(* Logix 5000 project; controller cal1632 1756-L62 rev 16.20; software revision 16.05; part 13 of 57 *)
(* tags used below, declared in another part *)
   AFI : BOOL;
   FAULT : BOOL;
   p01_param_fan_zero_speed : REAL;
   p01_param_open_oven_exh_sp : REAL;
   p01_param_open_oven_recirc_sp : REAL;
   p01_recipe_active : recipe;
   p01r02 : routine;
   p01r09_open_oven : BOOL;
   p01r09_pb_global_reset : BOOL;
   p02_dint_from_hmi : hmi_dint;
   p11_ai_exh_rpm : REAL;
   p11_ai_lfl : REAL;
   p11_ai_recirc_rpm : REAL;
   p11_ao_exhaust_selected_speed : REAL;
   p11_ao_recirc_selected_speed : REAL;
   p11_di_burner_auto : BOOL;
   p11_di_door_open : BOOL;
   p11_di_exh : acs800_di_normal;
   p11_di_exh_fan_mtr_ts : BOOL;
   p11_di_exh_flow_ok : BOOL;
   p11_di_flame_on : BOOL;
   p11_di_fresh_air_clean : BOOL;
   p11_di_recirc : acs800_di_normal;
   p11_di_recirc_fan_mtr_ts : BOOL;
   p11_di_recirc_flow_ok : BOOL;
   p11_di_sp00 : BOOL;
   p11_di_tc01_bo : BOOL;
   p11_di_tc02_bo : BOOL;
   p11_di_zone_air_clean : BOOL;
   p11_do_enable_burner : BOOL;
   p11_do_exh : acs800_do_normal;
   p11_do_recirc : acs800_do_normal;
   p11_param_lfl_hl : REAL;
   p11_param_tc01_dev : REAL;
   p11r02_shutdown_temp : BOOL;
   p11r20_safeties_ok : BOOL;
   p11r20_state : DINT;
   p11r30 : routine;
   p11r30_pb_zone_on : BOOL;
   p11r30_pid_temp_sp_error : REAL;
   p11r30_request_deviation_warning : BOOL;
   p11r30_request_heat : BOOL;
   p11r30_request_heat_last : BOOL;
   p11r30_request_manual : BOOL;
   p11r30_timer_fault : TIMER[16];
   p11r30_timer_warning : TIMER[12];
   p11r31 : routine;
   p11r31_pb_start : BOOL;
   p11r31_pb_stop : BOOL;
   p11r31_request_auto_run : BOOL;
   p11r31_run_permissive : BOOL;
   p11r31_timer_fault : TIMER[5];
   p11r31_timer_warning : TIMER[5];
   p11r31_vfd_stopped : BOOL;
   p11r32 : routine;
   p11r32_pb_start : BOOL;
   p11r32_pb_stop : BOOL;
   p11r32_request_auto_run : BOOL;
   p11r32_run_permissive : BOOL;
   p11r32_timer_fault : TIMER[5];
   p11r32_timer_warning : TIMER[5];
   p11r32_vfd_stopped : BOOL;
   p12r30 : routine;
   p23_di_exhaust_speed_ok : BOOL;
   p23_di_supply_speed_ok : BOOL;
   p23r02 : routine;
(* P11_Zone_1, continued *)

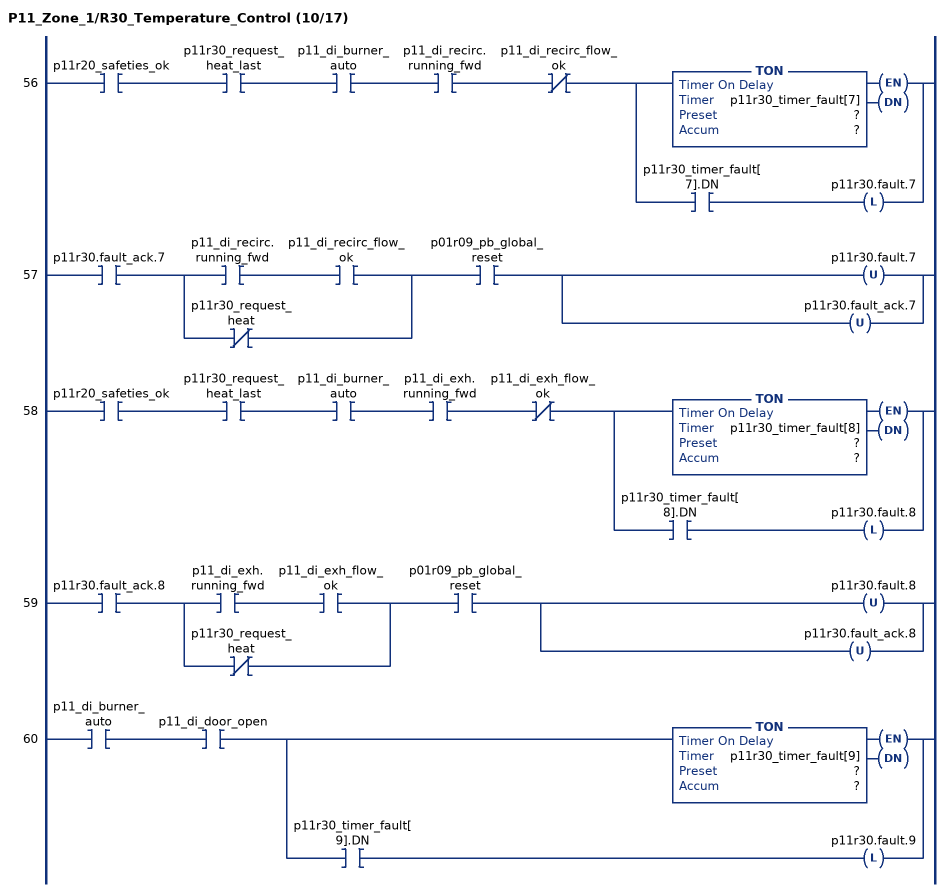
   [picture p239: P11_Zone_1/R30_Temperature_Control rungs 56-60]
   56: XIC(p11r20_safeties_ok)XIC(p11r30_request_heat_last)XIC(p11_di_burner_auto)XIC(p11_di_recirc.running_fwd)XIO(p11_di_recirc_flow_ok)[TON(p11r30_timer_fault[7],?,?) ,XIC(p11r30_timer_fault[7].DN) OTL(p11r30.fault.7) ];
   57: XIC(p11r30.fault_ack.7)[XIC(p11_di_recirc.running_fwd) XIC(p11_di_recirc_flow_ok) ,XIO(p11r30_request_heat) ]XIC(p01r09_pb_global_reset)[OTU(p11r30.fault.7) ,OTU(p11r30.fault_ack.7) ];
   58: XIC(p11r20_safeties_ok)XIC(p11r30_request_heat_last)XIC(p11_di_burner_auto)XIC(p11_di_exh.running_fwd)XIO(p11_di_exh_flow_ok)[TON(p11r30_timer_fault[8],?,?) ,XIC(p11r30_timer_fault[8].DN) OTL(p11r30.fault.8) ];
   59: XIC(p11r30.fault_ack.8)[XIC(p11_di_exh.running_fwd) XIC(p11_di_exh_flow_ok) ,XIO(p11r30_request_heat) ]XIC(p01r09_pb_global_reset)[OTU(p11r30.fault.8) ,OTU(p11r30.fault_ack.8) ];
   60: XIC(p11_di_burner_auto)XIC(p11_di_door_open)[TON(p11r30_timer_fault[9],?,?) ,XIC(p11r30_timer_fault[9].DN) OTL(p11r30.fault.9) ];
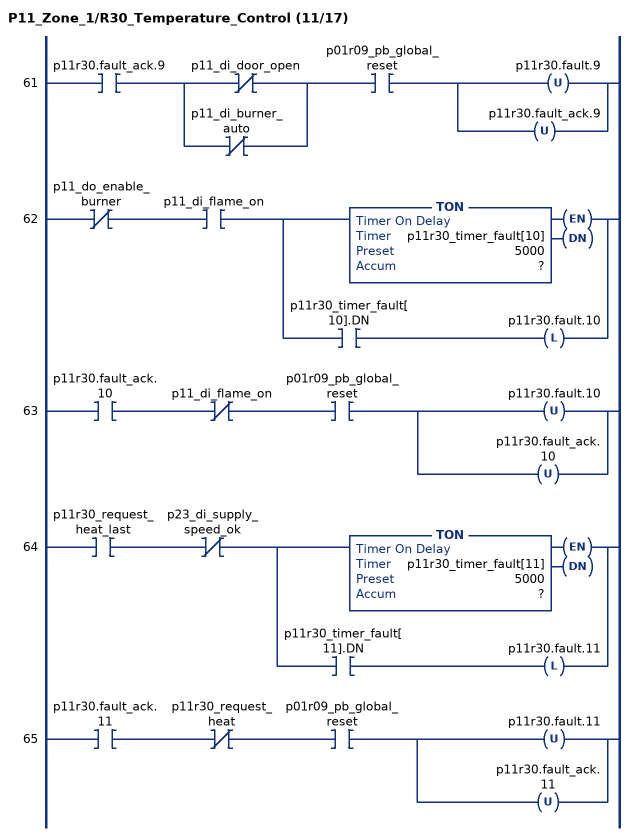
   61: XIC(p11r30.fault_ack.9)[XIO(p11_di_door_open) ,XIO(p11_di_burner_auto) ]XIC(p01r09_pb_global_reset)[OTU(p11r30.fault.9) ,OTU(p11r30.fault_ack.9) ];
   62: XIO(p11_do_enable_burner)XIC(p11_di_flame_on)[TON(p11r30_timer_fault[10],?,?) ,XIC(p11r30_timer_fault[10].DN) OTL(p11r30.fault.10) ];
   63: XIC(p11r30.fault_ack.10)XIO(p11_di_flame_on)XIC(p01r09_pb_global_reset)[OTU(p11r30.fault.10) ,OTU(p11r30.fault_ack.10) ];
   64: XIC(p11r30_request_heat_last)XIO(p23_di_supply_speed_ok)[TON(p11r30_timer_fault[11],?,?) ,XIC(p11r30_timer_fault[11].DN) OTL(p11r30.fault.11) ];
   65: XIC(p11r30.fault_ack.11)XIO(p11r30_request_heat)XIC(p01r09_pb_global_reset)[OTU(p11r30.fault.11) ,OTU(p11r30.fault_ack.11) ];
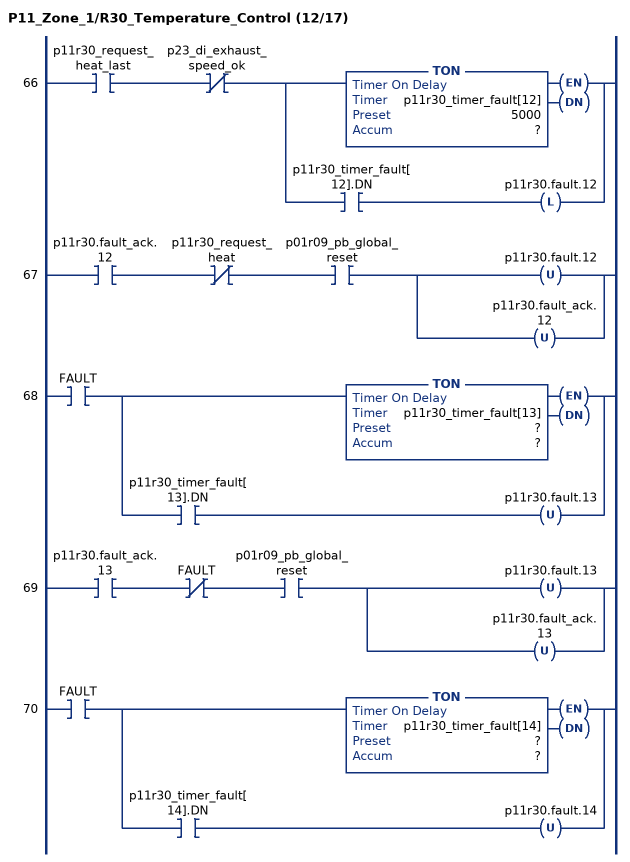
   66: XIC(p11r30_request_heat_last)XIO(p23_di_exhaust_speed_ok)[TON(p11r30_timer_fault[12],?,?) ,XIC(p11r30_timer_fault[12].DN) OTL(p11r30.fault.12) ];
   67: XIC(p11r30.fault_ack.12)XIO(p11r30_request_heat)XIC(p01r09_pb_global_reset)[OTU(p11r30.fault.12) ,OTU(p11r30.fault_ack.12) ];
   68: XIC(FAULT)[TON(p11r30_timer_fault[13],?,?) ,XIC(p11r30_timer_fault[13].DN) OTU(p11r30.fault.13) ];
   69: XIC(p11r30.fault_ack.13)XIO(FAULT)XIC(p01r09_pb_global_reset)[OTU(p11r30.fault.13) ,OTU(p11r30.fault_ack.13) ];
   70: XIC(FAULT)[TON(p11r30_timer_fault[14],?,?) ,XIC(p11r30_timer_fault[14].DN) OTU(p11r30.fault.14) ];
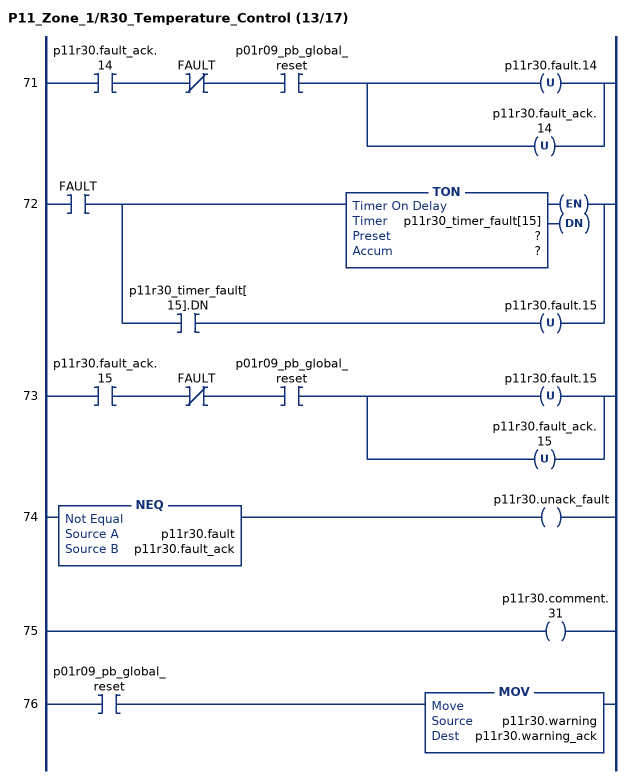
   71: XIC(p11r30.fault_ack.14)XIO(FAULT)XIC(p01r09_pb_global_reset)[OTU(p11r30.fault.14) ,OTU(p11r30.fault_ack.14) ];
   72: XIC(FAULT)[TON(p11r30_timer_fault[15],?,?) ,XIC(p11r30_timer_fault[15].DN) OTU(p11r30.fault.15) ];
   73: XIC(p11r30.fault_ack.15)XIO(FAULT)XIC(p01r09_pb_global_reset)[OTU(p11r30.fault.15) ,OTU(p11r30.fault_ack.15) ];
   74: NEQ(p11r30.fault,p11r30.fault_ack)OTE(p11r30.unack_fault);
   75: OTE(p11r30.comment.31);
   76: XIC(p01r09_pb_global_reset)MOV(p11r30.warning,p11r30.warning_ack);
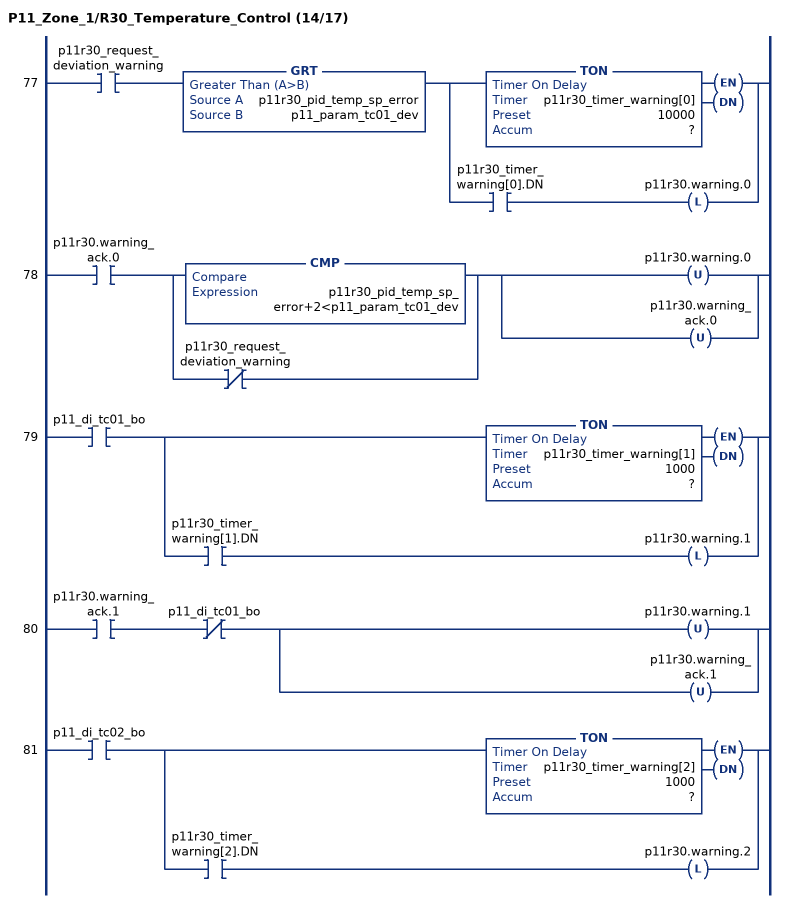
   77: XIC(p11r30_request_deviation_warning)GRT(p11r30_pid_temp_sp_error,p11_param_tc01_dev)[TON(p11r30_timer_warning[0],?,?) ,XIC(p11r30_timer_warning[0].DN) OTL(p11r30.warning.0) ];
   78: XIC(p11r30.warning_ack.0)[CMP(p11r30_pid_temp_sp_error+2<p11_param_tc01_dev) ,XIO(p11r30_request_deviation_warning) ][OTU(p11r30.warning.0) ,OTU(p11r30.warning_ack.0) ];
   79: XIC(p11_di_tc01_bo)[TON(p11r30_timer_warning[1],?,?) ,XIC(p11r30_timer_warning[1].DN) OTL(p11r30.warning.1) ];
   80: XIC(p11r30.warning_ack.1)XIO(p11_di_tc01_bo)[OTU(p11r30.warning.1) ,OTU(p11r30.warning_ack.1) ];
   81: XIC(p11_di_tc02_bo)[TON(p11r30_timer_warning[2],?,?) ,XIC(p11r30_timer_warning[2].DN) OTL(p11r30.warning.2) ];
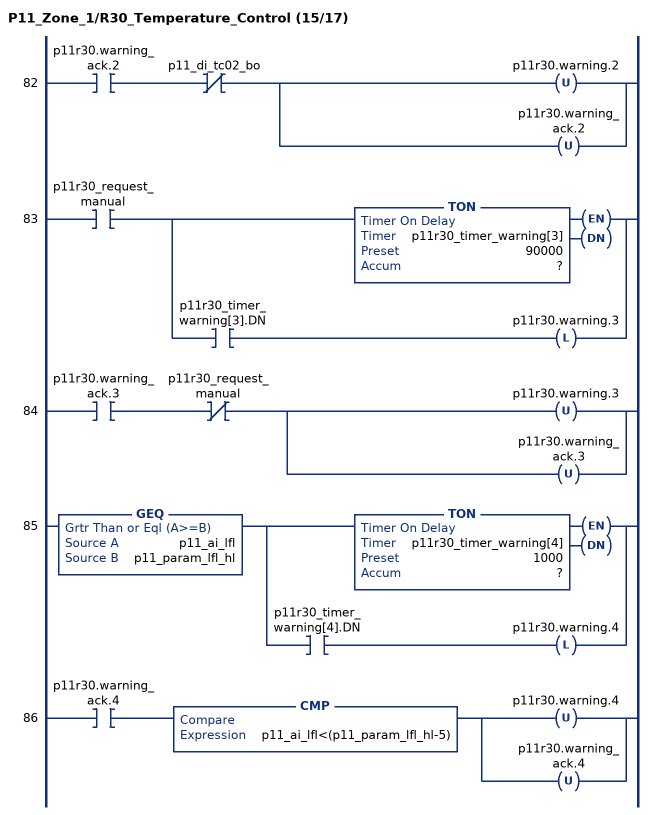
   82: XIC(p11r30.warning_ack.2)XIO(p11_di_tc02_bo)[OTU(p11r30.warning.2) ,OTU(p11r30.warning_ack.2) ];
   83: XIC(p11r30_request_manual)[TON(p11r30_timer_warning[3],?,?) ,XIC(p11r30_timer_warning[3].DN) OTL(p11r30.warning.3) ];
   84: XIC(p11r30.warning_ack.3)XIO(p11r30_request_manual)[OTU(p11r30.warning.3) ,OTU(p11r30.warning_ack.3) ];
   85: GEQ(p11_ai_lfl,p11_param_lfl_hl)[TON(p11r30_timer_warning[4],?,?) ,XIC(p11r30_timer_warning[4].DN) OTL(p11r30.warning.4) ];
   86: XIC(p11r30.warning_ack.4)CMP(p11_ai_lfl<(p11_param_lfl_hl-5))[OTU(p11r30.warning.4) ,OTU(p11r30.warning_ack.4) ];
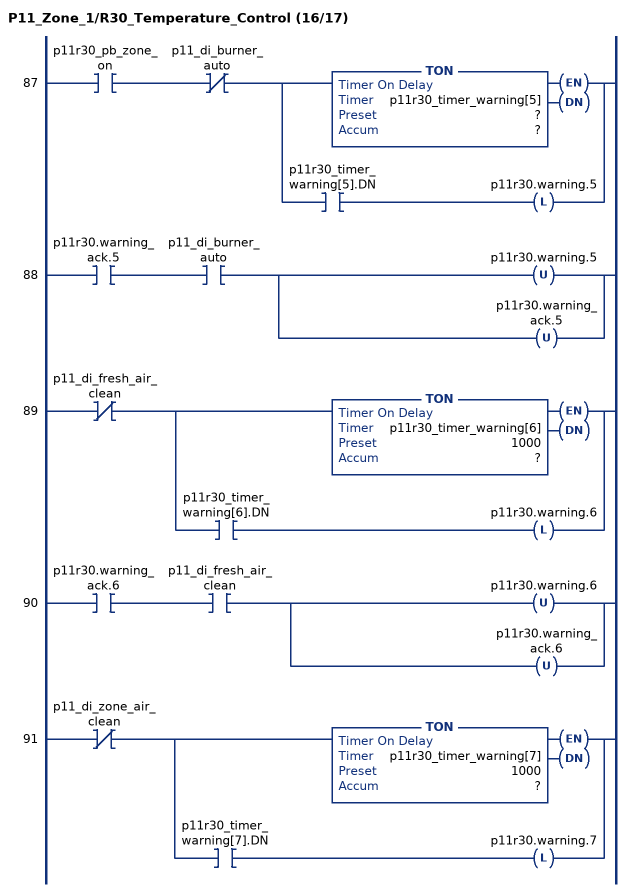
   87: XIC(p11r30_pb_zone_on)XIO(p11_di_burner_auto)[TON(p11r30_timer_warning[5],?,?) ,XIC(p11r30_timer_warning[5].DN) OTL(p11r30.warning.5) ];
   88: XIC(p11r30.warning_ack.5)XIC(p11_di_burner_auto)[OTU(p11r30.warning.5) ,OTU(p11r30.warning_ack.5) ];
   89: XIO(p11_di_fresh_air_clean)[TON(p11r30_timer_warning[6],?,?) ,XIC(p11r30_timer_warning[6].DN) OTL(p11r30.warning.6) ];
   90: XIC(p11r30.warning_ack.6)XIC(p11_di_fresh_air_clean)[OTU(p11r30.warning.6) ,OTU(p11r30.warning_ack.6) ];
   91: XIO(p11_di_zone_air_clean)[TON(p11r30_timer_warning[7],?,?) ,XIC(p11r30_timer_warning[7].DN) OTL(p11r30.warning.7) ];
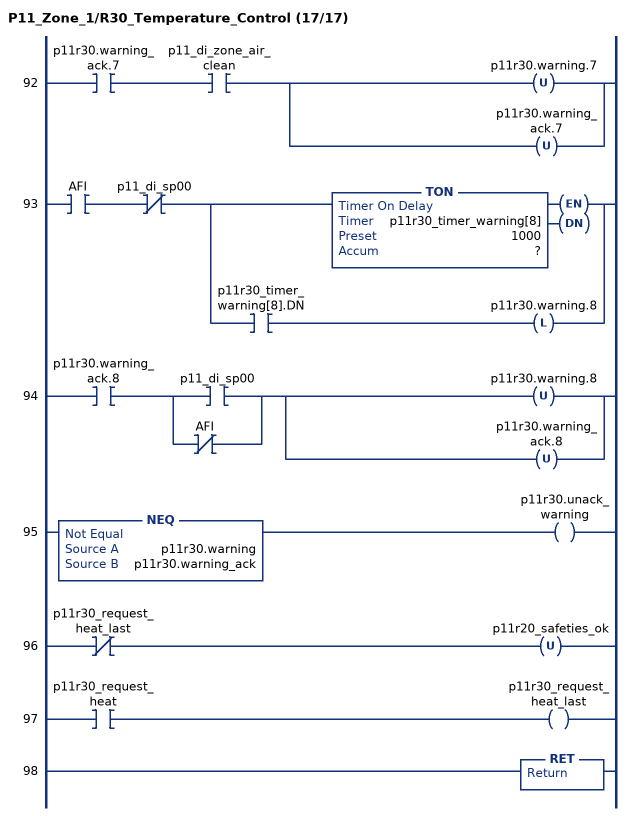
   92: XIC(p11r30.warning_ack.7)XIC(p11_di_zone_air_clean)[OTU(p11r30.warning.7) ,OTU(p11r30.warning_ack.7) ];
   93: XIC(AFI)XIO(p11_di_sp00)[TON(p11r30_timer_warning[8],?,?) ,XIC(p11r30_timer_warning[8].DN) OTL(p11r30.warning.8) ];
   94: XIC(p11r30.warning_ack.8)[XIC(p11_di_sp00) ,XIO(AFI) ][OTU(p11r30.warning.8) ,OTU(p11r30.warning_ack.8) ];
   95: NEQ(p11r30.warning,p11r30.warning_ack)OTE(p11r30.unack_warning);
   96: XIO(p11r30_request_heat_last)OTU(p11r20_safeties_ok);
   97: XIC(p11r30_request_heat)OTE(p11r30_request_heat_last);
   98: RET();
END_ROUTINE

ROUTINE R31_Exhaust_VFD   (* ladder *)
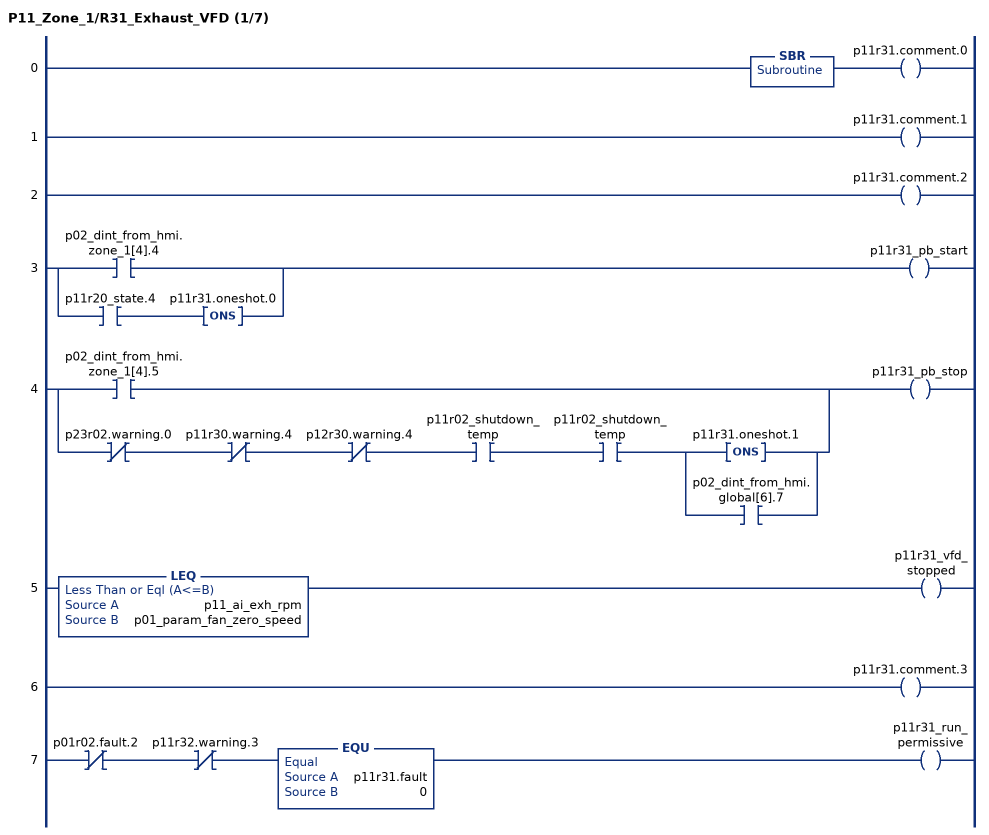
   0: SBR()OTE(p11r31.comment.0);
   1: OTE(p11r31.comment.1);
   2: OTE(p11r31.comment.2);
   3: [XIC(p02_dint_from_hmi.zone_1[4].4) ,XIC(p11r20_state.4) ONS(p11r31.oneshot.0) ]OTE(p11r31_pb_start);
   4: [XIC(p02_dint_from_hmi.zone_1[4].5) ,XIO(p23r02.warning.0) XIO(p11r30.warning.4) XIO(p12r30.warning.4) XIC(p11r02_shutdown_temp) XIC(p11r02_shutdown_temp) [ONS(p11r31.oneshot.1) ,XIC(p02_dint_from_hmi.global[6].7) ] ]OTE(p11r31_pb_stop);
   5: LEQ(p11_ai_exh_rpm,p01_param_fan_zero_speed)OTE(p11r31_vfd_stopped);
   6: OTE(p11r31.comment.3);
   7: XIO(p01r02.fault.2)XIO(p11r32.warning.3)EQU(p11r31.fault,0)OTE(p11r31_run_permissive);
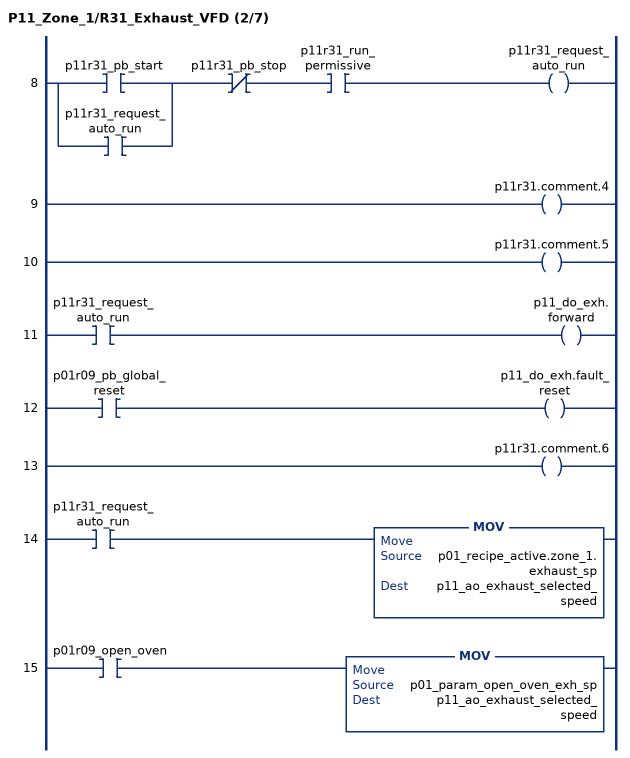
   8: [XIC(p11r31_pb_start) ,XIC(p11r31_request_auto_run) ]XIO(p11r31_pb_stop)XIC(p11r31_run_permissive)OTE(p11r31_request_auto_run);
   9: OTE(p11r31.comment.4);
   10: OTE(p11r31.comment.5);
   11: XIC(p11r31_request_auto_run)OTE(p11_do_exh.forward);
   12: XIC(p01r09_pb_global_reset)OTE(p11_do_exh.fault_reset);
   13: OTE(p11r31.comment.6);
   14: XIC(p11r31_request_auto_run)MOV(p01_recipe_active.zone_1.exhaust_sp,p11_ao_exhaust_selected_speed);
   15: XIC(p01r09_open_oven)MOV(p01_param_open_oven_exh_sp,p11_ao_exhaust_selected_speed);
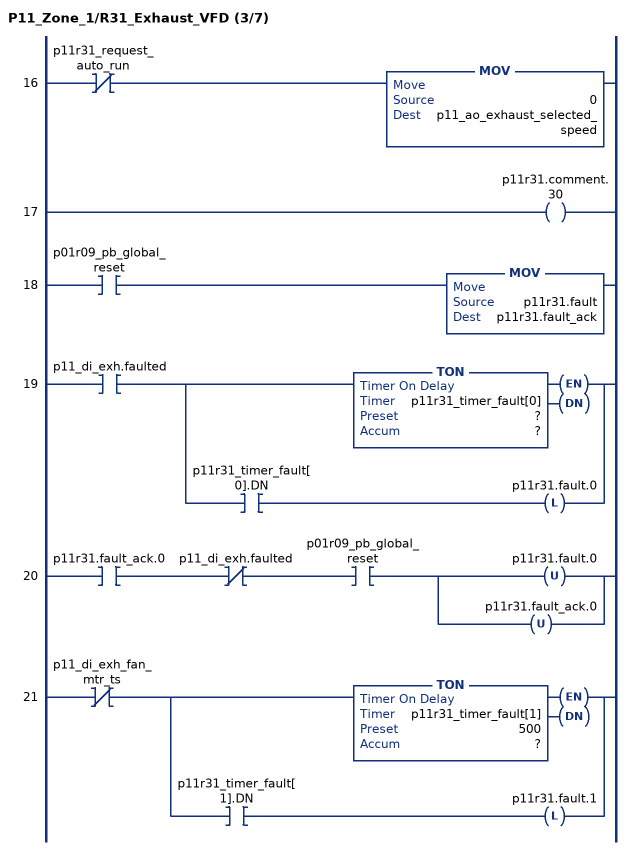
   16: XIO(p11r31_request_auto_run)MOV(0,p11_ao_exhaust_selected_speed);
   17: OTE(p11r31.comment.30);
   18: XIC(p01r09_pb_global_reset)MOV(p11r31.fault,p11r31.fault_ack);
   19: XIC(p11_di_exh.faulted)[TON(p11r31_timer_fault[0],?,?) ,XIC(p11r31_timer_fault[0].DN) OTL(p11r31.fault.0) ];
   20: XIC(p11r31.fault_ack.0)XIO(p11_di_exh.faulted)XIC(p01r09_pb_global_reset)[OTU(p11r31.fault.0) ,OTU(p11r31.fault_ack.0) ];
   21: XIO(p11_di_exh_fan_mtr_ts)[TON(p11r31_timer_fault[1],?,?) ,XIC(p11r31_timer_fault[1].DN) OTL(p11r31.fault.1) ];
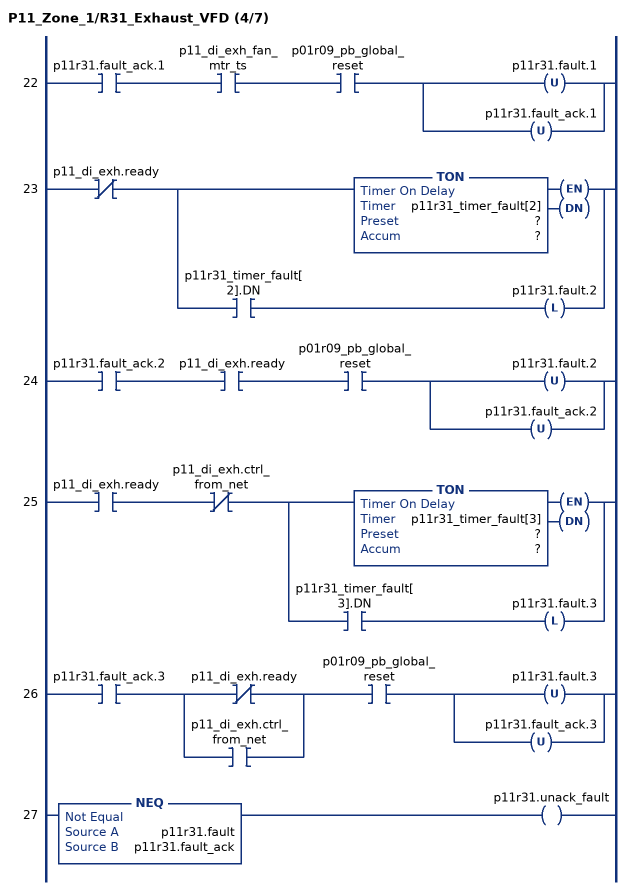
   22: XIC(p11r31.fault_ack.1)XIC(p11_di_exh_fan_mtr_ts)XIC(p01r09_pb_global_reset)[OTU(p11r31.fault.1) ,OTU(p11r31.fault_ack.1) ];
   23: XIO(p11_di_exh.ready)[TON(p11r31_timer_fault[2],?,?) ,XIC(p11r31_timer_fault[2].DN) OTL(p11r31.fault.2) ];
   24: XIC(p11r31.fault_ack.2)XIC(p11_di_exh.ready)XIC(p01r09_pb_global_reset)[OTU(p11r31.fault.2) ,OTU(p11r31.fault_ack.2) ];
   25: XIC(p11_di_exh.ready)XIO(p11_di_exh.ctrl_from_net)[TON(p11r31_timer_fault[3],?,?) ,XIC(p11r31_timer_fault[3].DN) OTL(p11r31.fault.3) ];
   26: XIC(p11r31.fault_ack.3)[XIO(p11_di_exh.ready) ,XIC(p11_di_exh.ctrl_from_net) ]XIC(p01r09_pb_global_reset)[OTU(p11r31.fault.3) ,OTU(p11r31.fault_ack.3) ];
   27: NEQ(p11r31.fault,p11r31.fault_ack)OTE(p11r31.unack_fault);
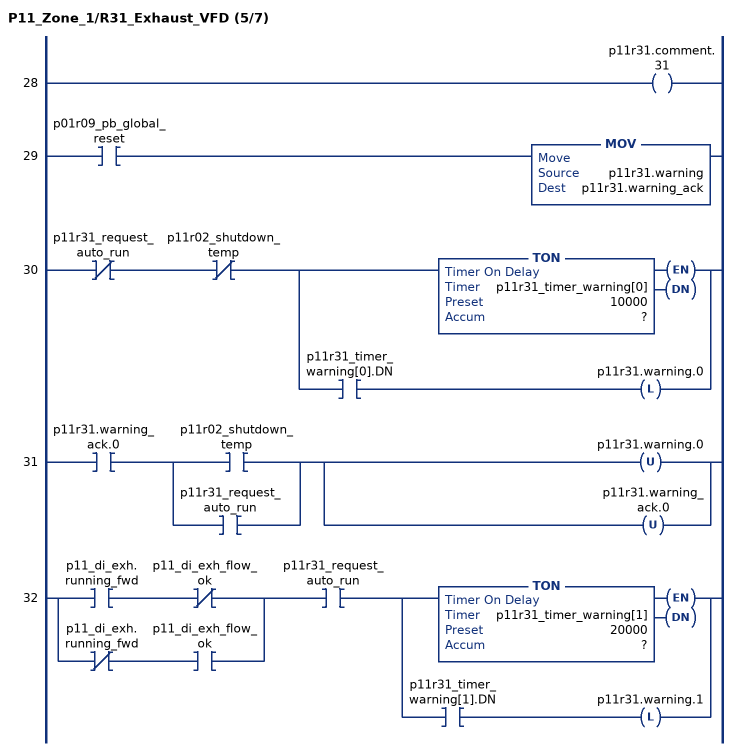
   28: OTE(p11r31.comment.31);
   29: XIC(p01r09_pb_global_reset)MOV(p11r31.warning,p11r31.warning_ack);
   30: XIO(p11r31_request_auto_run)XIO(p11r02_shutdown_temp)[TON(p11r31_timer_warning[0],?,?) ,XIC(p11r31_timer_warning[0].DN) OTL(p11r31.warning.0) ];
   31: XIC(p11r31.warning_ack.0)[XIC(p11r02_shutdown_temp) ,XIC(p11r31_request_auto_run) ][OTU(p11r31.warning.0) ,OTU(p11r31.warning_ack.0) ];
   32: [XIC(p11_di_exh.running_fwd) XIO(p11_di_exh_flow_ok) ,XIO(p11_di_exh.running_fwd) XIC(p11_di_exh_flow_ok) ]XIC(p11r31_request_auto_run)[TON(p11r31_timer_warning[1],?,?) ,XIC(p11r31_timer_warning[1].DN) OTL(p11r31.warning.1) ];
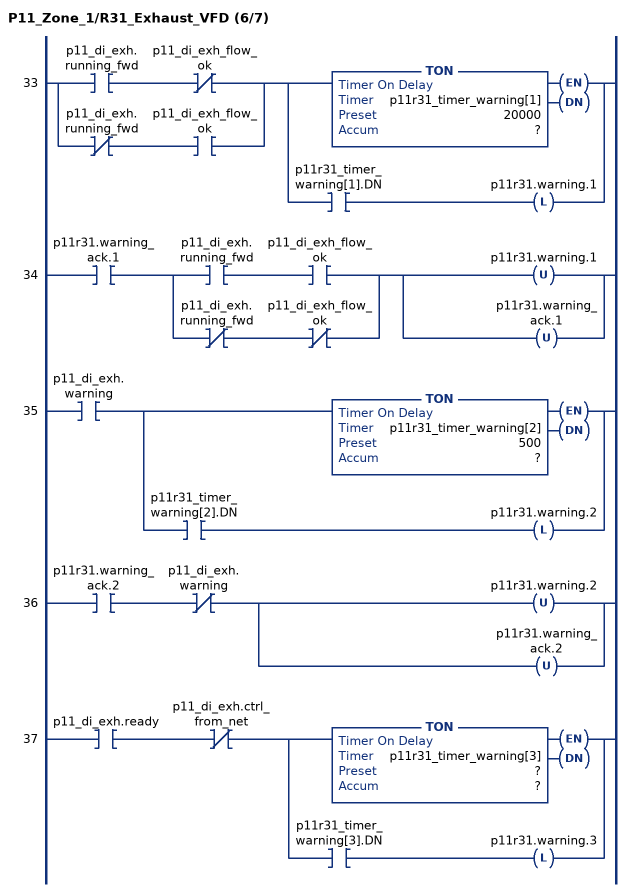
   33: [XIC(p11_di_exh.running_fwd) XIO(p11_di_exh_flow_ok) ,XIO(p11_di_exh.running_fwd) XIC(p11_di_exh_flow_ok) ][TON(p11r31_timer_warning[1],?,?) ,XIC(p11r31_timer_warning[1].DN) OTL(p11r31.warning.1) ];
   34: XIC(p11r31.warning_ack.1)[XIC(p11_di_exh.running_fwd) XIC(p11_di_exh_flow_ok) ,XIO(p11_di_exh.running_fwd) XIO(p11_di_exh_flow_ok) ][OTU(p11r31.warning.1) ,OTU(p11r31.warning_ack.1) ];
   35: XIC(p11_di_exh.warning)[TON(p11r31_timer_warning[2],?,?) ,XIC(p11r31_timer_warning[2].DN) OTL(p11r31.warning.2) ];
   36: XIC(p11r31.warning_ack.2)XIO(p11_di_exh.warning)[OTU(p11r31.warning.2) ,OTU(p11r31.warning_ack.2) ];
   37: XIC(p11_di_exh.ready)XIO(p11_di_exh.ctrl_from_net)[TON(p11r31_timer_warning[3],?,?) ,XIC(p11r31_timer_warning[3].DN) OTL(p11r31.warning.3) ];
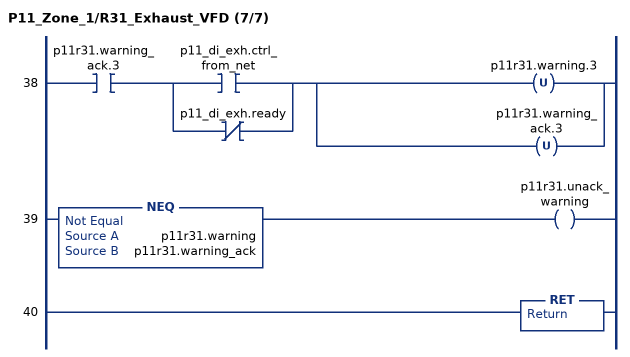
   38: XIC(p11r31.warning_ack.3)[XIC(p11_di_exh.ctrl_from_net) ,XIO(p11_di_exh.ready) ][OTU(p11r31.warning.3) ,OTU(p11r31.warning_ack.3) ];
   39: NEQ(p11r31.warning,p11r31.warning_ack)OTE(p11r31.unack_warning);
   40: RET();
END_ROUTINE

ROUTINE R32_Recirc_VFD   (* ladder *)
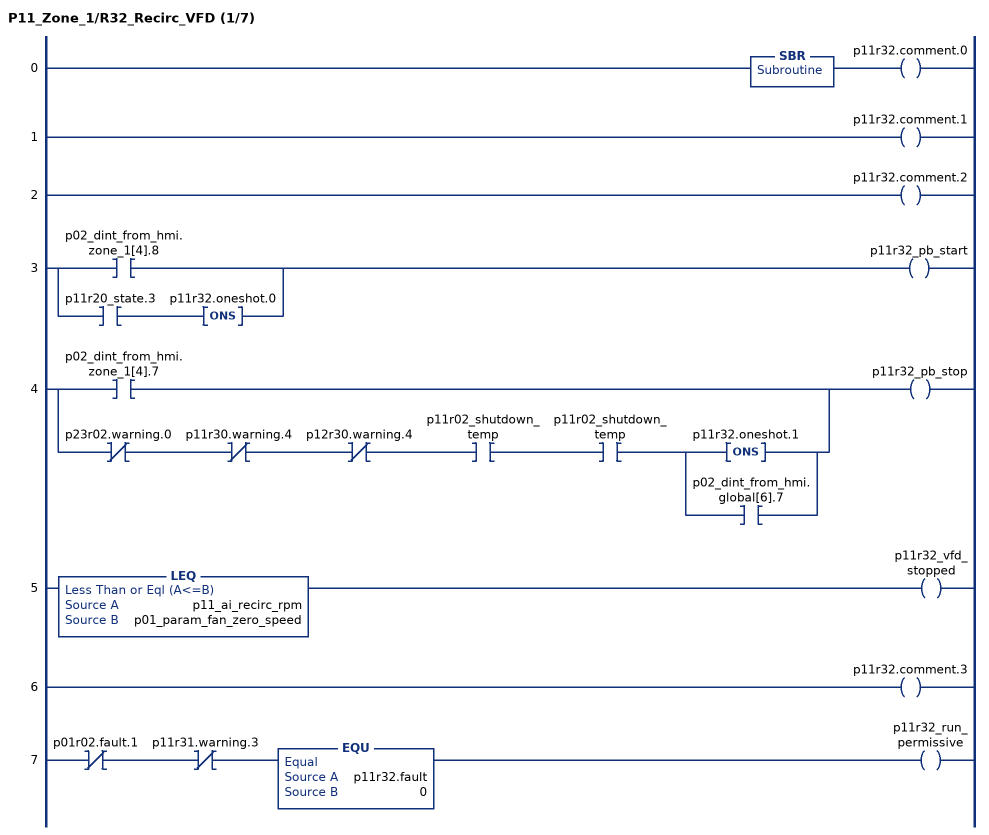
   0: SBR()OTE(p11r32.comment.0);
   1: OTE(p11r32.comment.1);
   2: OTE(p11r32.comment.2);
   3: [XIC(p02_dint_from_hmi.zone_1[4].8) ,XIC(p11r20_state.3) ONS(p11r32.oneshot.0) ]OTE(p11r32_pb_start);
   4: [XIC(p02_dint_from_hmi.zone_1[4].7) ,XIO(p23r02.warning.0) XIO(p11r30.warning.4) XIO(p12r30.warning.4) XIC(p11r02_shutdown_temp) XIC(p11r02_shutdown_temp) [ONS(p11r32.oneshot.1) ,XIC(p02_dint_from_hmi.global[6].7) ] ]OTE(p11r32_pb_stop);
   5: LEQ(p11_ai_recirc_rpm,p01_param_fan_zero_speed)OTE(p11r32_vfd_stopped);
   6: OTE(p11r32.comment.3);
   7: XIO(p01r02.fault.1)XIO(p11r31.warning.3)EQU(p11r32.fault,0)OTE(p11r32_run_permissive);
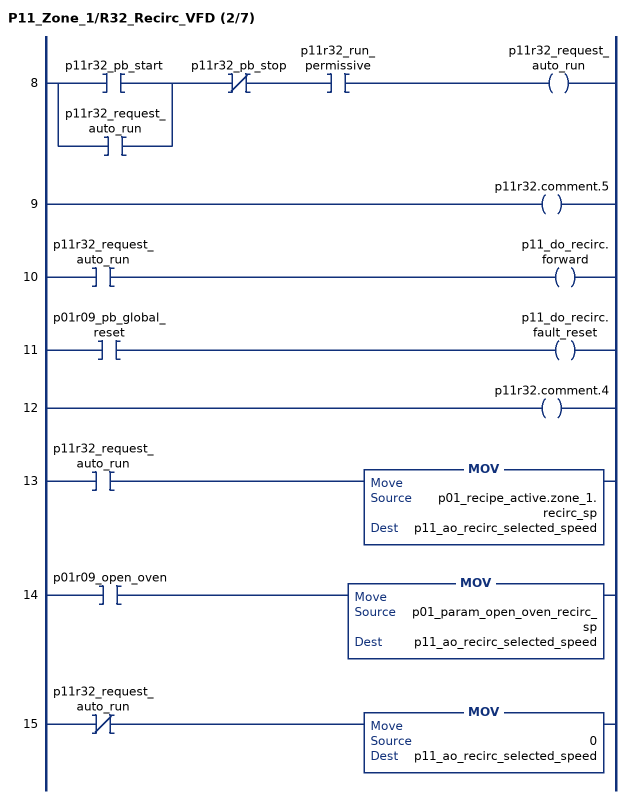
   8: [XIC(p11r32_pb_start) ,XIC(p11r32_request_auto_run) ]XIO(p11r32_pb_stop)XIC(p11r32_run_permissive)OTE(p11r32_request_auto_run);
   9: OTE(p11r32.comment.5);
   10: XIC(p11r32_request_auto_run)OTE(p11_do_recirc.forward);
   11: XIC(p01r09_pb_global_reset)OTE(p11_do_recirc.fault_reset);
   12: OTE(p11r32.comment.4);
   13: XIC(p11r32_request_auto_run)MOV(p01_recipe_active.zone_1.recirc_sp,p11_ao_recirc_selected_speed);
   14: XIC(p01r09_open_oven)MOV(p01_param_open_oven_recirc_sp,p11_ao_recirc_selected_speed);
   15: XIO(p11r32_request_auto_run)MOV(0,p11_ao_recirc_selected_speed);
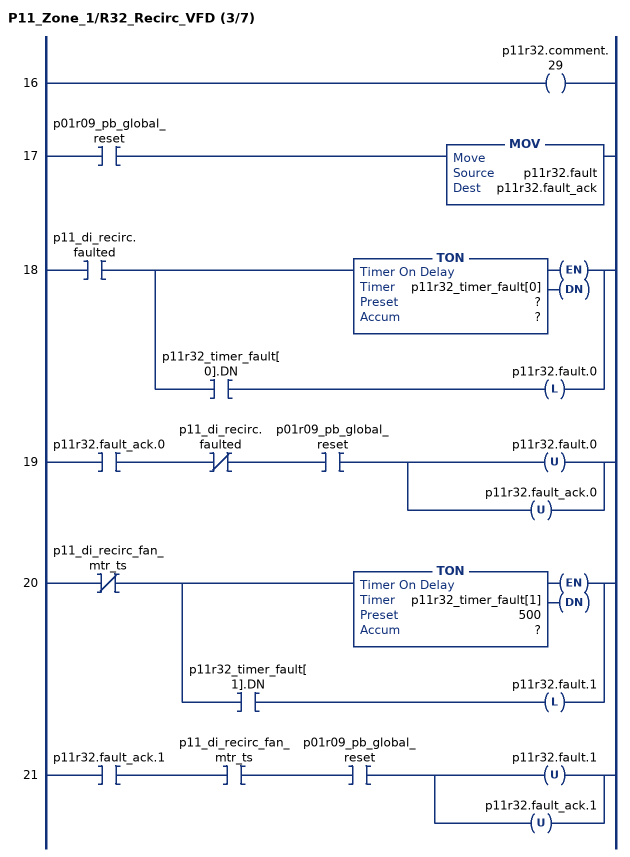
   16: OTE(p11r32.comment.29);
   17: XIC(p01r09_pb_global_reset)MOV(p11r32.fault,p11r32.fault_ack);
   18: XIC(p11_di_recirc.faulted)[TON(p11r32_timer_fault[0],?,?) ,XIC(p11r32_timer_fault[0].DN) OTL(p11r32.fault.0) ];
   19: XIC(p11r32.fault_ack.0)XIO(p11_di_recirc.faulted)XIC(p01r09_pb_global_reset)[OTU(p11r32.fault.0) ,OTU(p11r32.fault_ack.0) ];
   20: XIO(p11_di_recirc_fan_mtr_ts)[TON(p11r32_timer_fault[1],?,?) ,XIC(p11r32_timer_fault[1].DN) OTL(p11r32.fault.1) ];
   21: XIC(p11r32.fault_ack.1)XIC(p11_di_recirc_fan_mtr_ts)XIC(p01r09_pb_global_reset)[OTU(p11r32.fault.1) ,OTU(p11r32.fault_ack.1) ];
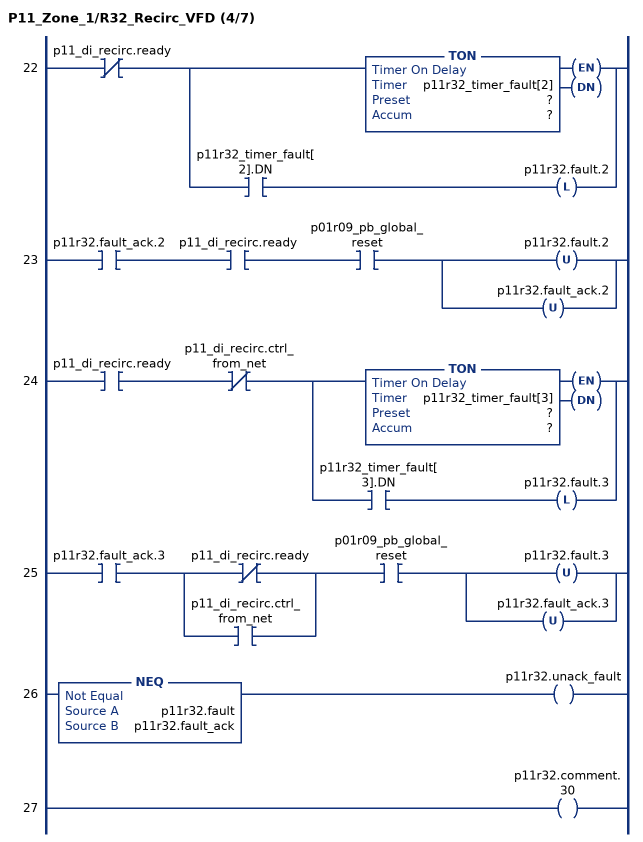
   22: XIO(p11_di_recirc.ready)[TON(p11r32_timer_fault[2],?,?) ,XIC(p11r32_timer_fault[2].DN) OTL(p11r32.fault.2) ];
   23: XIC(p11r32.fault_ack.2)XIC(p11_di_recirc.ready)XIC(p01r09_pb_global_reset)[OTU(p11r32.fault.2) ,OTU(p11r32.fault_ack.2) ];
   24: XIC(p11_di_recirc.ready)XIO(p11_di_recirc.ctrl_from_net)[TON(p11r32_timer_fault[3],?,?) ,XIC(p11r32_timer_fault[3].DN) OTL(p11r32.fault.3) ];
   25: XIC(p11r32.fault_ack.3)[XIO(p11_di_recirc.ready) ,XIC(p11_di_recirc.ctrl_from_net) ]XIC(p01r09_pb_global_reset)[OTU(p11r32.fault.3) ,OTU(p11r32.fault_ack.3) ];
   26: NEQ(p11r32.fault,p11r32.fault_ack)OTE(p11r32.unack_fault);
   27: OTE(p11r32.comment.30);
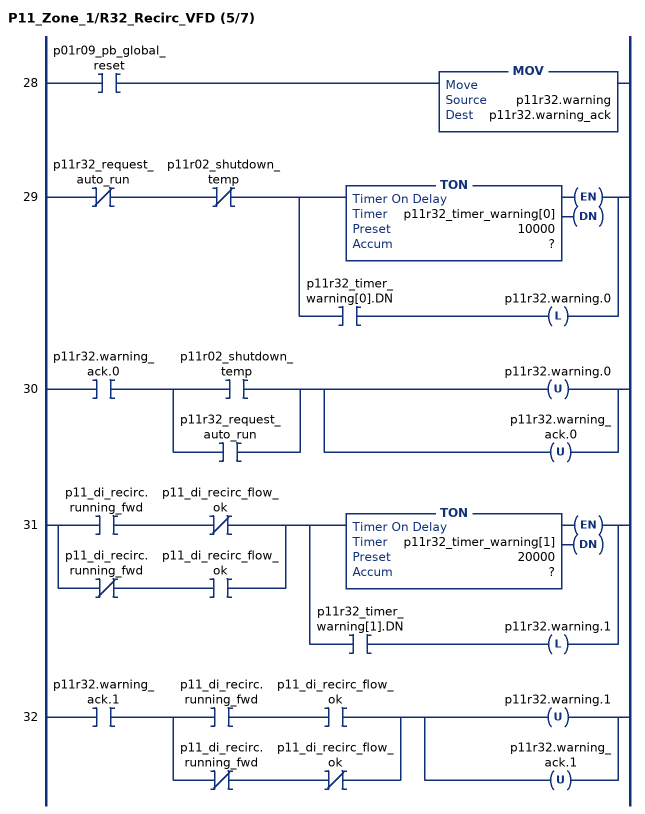
   28: XIC(p01r09_pb_global_reset)MOV(p11r32.warning,p11r32.warning_ack);
   29: XIO(p11r32_request_auto_run)XIO(p11r02_shutdown_temp)[TON(p11r32_timer_warning[0],?,?) ,XIC(p11r32_timer_warning[0].DN) OTL(p11r32.warning.0) ];
   30: XIC(p11r32.warning_ack.0)[XIC(p11r02_shutdown_temp) ,XIC(p11r32_request_auto_run) ][OTU(p11r32.warning.0) ,OTU(p11r32.warning_ack.0) ];
   31: [XIC(p11_di_recirc.running_fwd) XIO(p11_di_recirc_flow_ok) ,XIO(p11_di_recirc.running_fwd) XIC(p11_di_recirc_flow_ok) ][TON(p11r32_timer_warning[1],?,?) ,XIC(p11r32_timer_warning[1].DN) OTL(p11r32.warning.1) ];
   32: XIC(p11r32.warning_ack.1)[XIC(p11_di_recirc.running_fwd) XIC(p11_di_recirc_flow_ok) ,XIO(p11_di_recirc.running_fwd) XIO(p11_di_recirc_flow_ok) ][OTU(p11r32.warning.1) ,OTU(p11r32.warning_ack.1) ];
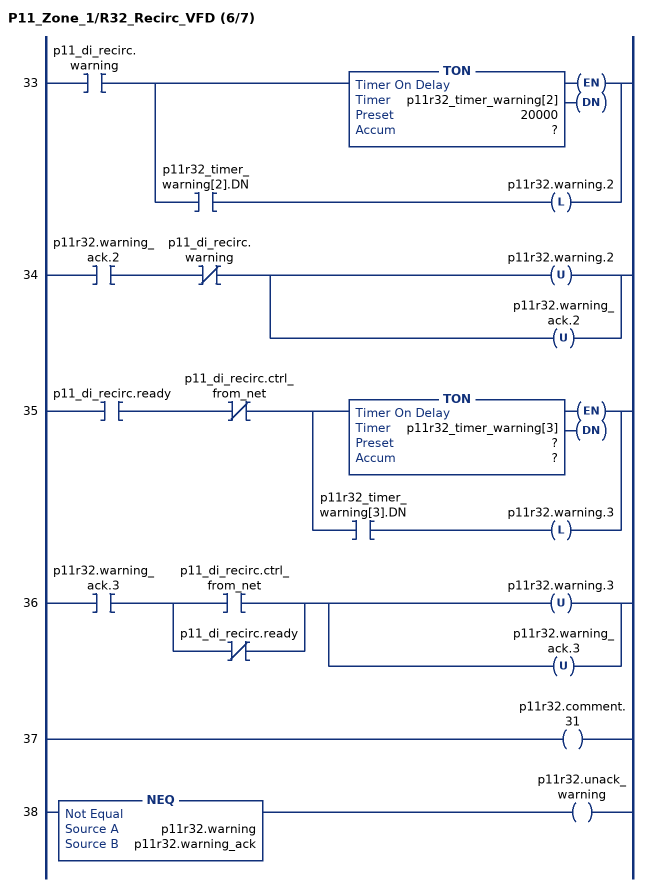
   33: XIC(p11_di_recirc.warning)[TON(p11r32_timer_warning[2],?,?) ,XIC(p11r32_timer_warning[2].DN) OTL(p11r32.warning.2) ];
   34: XIC(p11r32.warning_ack.2)XIO(p11_di_recirc.warning)[OTU(p11r32.warning.2) ,OTU(p11r32.warning_ack.2) ];
   35: XIC(p11_di_recirc.ready)XIO(p11_di_recirc.ctrl_from_net)[TON(p11r32_timer_warning[3],?,?) ,XIC(p11r32_timer_warning[3].DN) OTL(p11r32.warning.3) ];
   36: XIC(p11r32.warning_ack.3)[XIC(p11_di_recirc.ctrl_from_net) ,XIO(p11_di_recirc.ready) ][OTU(p11r32.warning.3) ,OTU(p11r32.warning_ack.3) ];
   37: OTE(p11r32.comment.31);
   38: NEQ(p11r32.warning,p11r32.warning_ack)OTE(p11r32.unack_warning);
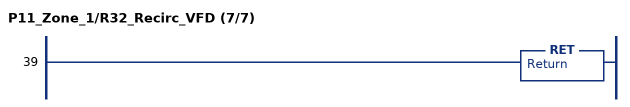
   39: RET();
END_ROUTINE
END_PROGRAM
